// TwinCAT 3 PLC project _3d_printer
// ProgramVersion: 3.1.4023.0
// libraries:
//   Tc2_MC2, * (Beckhoff Automation GmbH)
//   Tc2_NCI, * (Beckhoff Automation GmbH)
//   Tc2_NcKinematicTransformation, * (Beckhoff Automation GmbH)
//   Tc2_PlcInterpolation, * (Beckhoff Automation GmbH)
//   Tc2_Standard, * (Beckhoff Automation GmbH)
//   Tc2_System, * (Beckhoff Automation GmbH)
//   Tc3_Module, * (Beckhoff Automation GmbH)
// project tree:
//   / PlcTask.TcTTO
//   POUs/ FB_PowerChannel.TcPOU, MAIN.TcPOU
// real-time tasks:
//   TASK PlcTask: cycle T#10ms, priority 20, ADS port 350
// motion (NC):
//   TASK NC-Task 1 SAF: cycle T#2ms, priority 4, ADS port 501
//   TASK NC-Task 1 SVB: cycle T#10ms, priority 8, ADS port 511
//   AXIS axis xy 1 (id 1)
//     Dynamic: AccelerationMaximum=2000, DecelerationMaximum=2000, Acceleration=1000, Deceleration=1000
//     Velo: SlowManual=50, FastManual=100, Maximum=500
//     OtherSettings: AllowMotionCmdToSlave=true
//     encoder EncType=1
//       EncPara: ScaleFactorNumerator=40, ScaleFactorDenominator=12800
//         Inc: RefSoftSyncMask=#x0000ffff
//     drive DrvType=5
//       Analog: VeloReferenz=400, TorqueSetpointScale=10, ScaleFactorActTorque=0.1
//       TimeComp: TaskDelayCycles=1
//     controller CtrType=1
//       CtrPara: PriorControlFactor=1
//         Observer: BandWidth=20
//   AXIS axis xy 2 (id 2)
//     Dynamic: AccelerationMaximum=2000, DecelerationMaximum=2000, Acceleration=1000, Deceleration=1000
//     Velo: SlowManual=50, FastManual=100, Maximum=500
//     OtherSettings: AllowMotionCmdToSlave=true
//     encoder EncType=1
//       EncPara: ScaleFactorNumerator=40, ScaleFactorDenominator=12800
//         Inc: RefSoftSyncMask=#x0000ffff
//     drive DrvType=5
//       Analog: VeloReferenz=400, TorqueSetpointScale=10, ScaleFactorActTorque=0.1
//       TimeComp: TaskDelayCycles=1
//     controller CtrType=1
//       CtrPara: PriorControlFactor=1
//         Observer: BandWidth=20
//   AXIS Extruder (id 4)
//     Dynamic: AccelerationMaximum=100, DecelerationMaximum=100, Acceleration=100, Deceleration=100, Jerk=500
//     Velo: Maximum=10
//     OtherSettings: AllowMotionCmdToSlave=true
//     encoder EncType=1
//       EncPara: ScaleFactorNumerator=22.857, ScaleFactorDenominator=12800
//         Inc: RefSoftSyncMask=#x0000ffff
//     drive DrvType=5
//       Analog: VeloReferenz=5, TorqueSetpointScale=10, ScaleFactorActTorque=0.1
//       TimeComp: TaskDelayCycles=1
//     controller CtrType=1
//       CtrPara: PriorControlFactor=1
//         Observer: BandWidth=20
//   AXIS X axis (id 5)
//     Dynamic: AccelerationMaximum=2000, DecelerationMaximum=2000, Acceleration=1000, Deceleration=1000
//     Velo: SlowManual=50, FastManual=100, Maximum=500
//     OtherSettings: AllowMotionCmdToSlave=true
//     encoder EncType=1
//       EncPara: ScaleFactorNumerator=1, ScaleFactorDenominator=0.1
//     drive DrvType=5
//       Analog: VeloReferenz=500, TorqueSetpointScale=10, ScaleFactorActTorque=0.1
//       TimeComp: TaskDelayCycles=1
//     controller CtrType=1
//       CtrPara: PriorControlFactor=1
//         Observer: BandWidth=20
//   AXIS Z axis (id 3)
//     Dynamic: AccelerationMaximum=100, DecelerationMaximum=100, Acceleration=50, Deceleration=50, Jerk=1000
//     Velo: SlowManual=1, FastManual=5, Maximum=10
//     OtherSettings: AllowMotionCmdToSlave=true
//     encoder EncType=4
//       EncPara: ScaleFactorNumerator=8, ScaleFactorDenominator=12800, MaxCount=#x0000ffff
//         Inc: RefSoftSyncMask=#x0000ffff
//     drive DrvType=24
//       Analog: VeloReferenz=80, TorqueSetpointScale=10, ScaleFactorActTorque=0.1
//       TimeComp: TaskDelayCycles=1
//     controller CtrType=1
//       CtrPara: PriorControlFactor=1
//         Observer: BandWidth=20
//   AXIS Y axis (id 6)
//     Dynamic: AccelerationMaximum=2000, DecelerationMaximum=2000, Acceleration=1000, Deceleration=1000
//     Velo: SlowManual=50, FastManual=100, Maximum=500
//     OtherSettings: AllowMotionCmdToSlave=true
//     encoder EncType=1
//     drive DrvType=5
//       Analog: VeloReferenz=500, TorqueSetpointScale=10, ScaleFactorActTorque=0.1
//       TimeComp: TaskDelayCycles=1
//     controller CtrType=1
//       CtrPara: PriorControlFactor=1
//         Observer: BandWidth=20

CONFIGURATION _3d_printer
    RESOURCE PLC ON TwinCAT3
        TASK PlcTask(INTERVAL := T#10ms, PRIORITY := 20);
        PROGRAM MAIN WITH PlcTask : MAIN;
    END_RESOURCE
END_CONFIGURATION

// ---- POUs/MAIN.TcPOU
PROGRAM MAIN
VAR
	
	fbPower: FB_PowerChannel;
	runGCode: ItpEnableDefaultGCode;
	fbBuildGroup: CfgBuildExt3DGroup;
	fbLoadGCode: ItpLoadProgEx;
	fbStartGCode: ItpStartStopEx;
	fbConfirmHsk: ItpConfirmHsk;
	//getSParam :ItpGetSParam;
	
	fbConfigKinGroup: FB_KinConfigGroup;
    stAxesConfig: ST_KinAxes;
	in_stKinToPlc AT %I*  : NCTOPLC_NCICHANNEL_REF;
	
	Xaxis: AXIS_REF;
	Yaxis: AXIS_REF;
	Zaxis: AXIS_REF;
	Extruder: AXIS_REF;
	XY_1: AXIS_REF;
	XY_2: AXIS_REF;

	Xhome: MC_Home;
	Yhome: MC_Home;
	Zhome: MC_Home;
	
	Xjog: MC_Jog;
	Yjog: MC_Jog;
	
	HomingSensorX AT %I*: BOOL;
	HomingSensorY AT %I*: BOOL;
	HomingSensorZ AT %I*: BOOL;
	
	
	in_stNciToPlc AT %I*: NCTOPLC_NCICHANNEL_REF;
	out_stPlcToNci AT %Q*: PLCTONC_NCICHANNEL_REF;
	
	
	State: INT;
	bConfirmHsk: BOOL := FALSE;
	sPrgName: STRING(255) := 'test.txt';
	nInterpreterState: UDINT;
	
	bEnable: BOOL := TRUE;
END_VAR


fbPower(
	bEnable:=bEnable, 
	fOvr:= 100.0, 
	stX:=Xaxis, 
	stY:=Yaxis, 
	stZ:=Zaxis,
	stXY_1:= XY_1,
	stXY_2:= XY_2,
	stPlcToNci:=out_stPlcToNci , 
	bAllAxesReady=> );
	

	
CASE State OF
	0: // init
	
	IF fbPower.bAllAxesReady THEN
		State := 10; 
	END_IF
	
	10:
	
	stAxesConfig.nAxisIdsAcs[1] := XY_2.NcToPlc.AxisId;
	stAxesConfig.nAxisIdsAcs[2] := XY_1.NcToPlc.AxisId;
	stAxesConfig.nAxisIdsMcs[1] := Xaxis.NcToPlc.AxisId;
	stAxesConfig.nAxisIdsMcs[2] := Yaxis.NcToPlc.AxisId;
	
	fbConfigKinGroup(
    bExecute       := TRUE ,
    bCartesianMode := TRUE ,
    stAxesList     := stAxesConfig,
    stKinRefIn     := in_stKinToPlc );
	
	IF NOT fbConfigKinGroup.bBusy THEN
		IF NOT fbConfigKinGroup.bError THEN
			State:=20;
		END_IF
	END_IF
	20:
	Xjog(Axis:= Xaxis,JogBackwards:= TRUE , Velocity:= 0.01, Deceleration:= 1500);
	IF NOT HomingSensorX THEN
		Xjog(Axis:= Xaxis,JogBackwards:= FALSE);
		//State:=21;
	END_IF
	
	21:
	Yjog(Axis:= Yaxis,JogBackwards:= TRUE , Velocity:= 0.01, Deceleration:= 1500);
	IF NOT HomingSensorY THEN
		Yjog(Axis:= Yaxis,JogBackwards:= FALSE);
		
		//State:=21;
	END_IF
	
	22:
	Zhome(axis := Zaxis,execute := TRUE,BCalibrationCam := NOT HomingSensorZ);
	IF Zhome.Done THEN
		//State:=30;
	END_IF
	
	30:
	
	fbLoadGCode(
		sNciToPlc:=in_stNciToPlc, 
		bExecute:=TRUE, 
		sPrg:= sPrgName, 
		nLength:= INT_TO_UDINT(LEN(sPrgName)), 
		tTimeOut:= , 
		bBusy=> , 
		bErr=> , 
		nErrId=> );
	IF NOT fbLoadGCode.bBusy THEN
		IF NOT fbLoadGCode.bErr THEN
			fbLoadGCode(sNciToPlc:=in_stNciToPlc, bExecute:=FALSE); 
			State	:= 40;				
		END_IF
	END_IF
	40:
	
	nInterpreterState	:= ItpGetStateInterpreter(sNciToPlc:=in_stNciToPlc);
	IF nInterpreterState = Tc2_NCI.NCI_INTERPRETER_READY THEN
		State	:= 50;		
	END_IF
	50:
	fbBuildGroup(
		bExecute:=TRUE,
		nGroupId:=ItpGetGroupId(sNciToPlc:=in_stNciToPlc),
		nXAxisId:=XAxis.NcToPlc.AxisId,
		nYAxisId:=YAxis.NcToPlc.AxisId,
		nZAxisId:=ZAxis.NcToPlc.AxisId,
		tTimeOut:=T#2S );
		
	IF NOT fbBuildGroup.bBusy THEN
		fbBuildGroup( bExecute:=FALSE );
		
		IF NOT fbBuildGroup.bErr THEN
			State	:= 30;
		END_IF
	END_IF

	
	60:
	
	// start g-code file
	fbStartGCode(
		bStart:=TRUE, 
		bStop:=FALSE, 
		tTimeOut:= , 
		sNciToPlc:= in_stNciToPlc, 
		bBusy=> , 
		bErr=> , 
		nErrId=> );
	IF NOT fbStartGCode.bBusy THEN
		IF NOT fbStartGCode.bErr THEN
			State	:= 60;			
		END_IF
		fbStartGCode( bStart:=FALSE, sNciToPlc:= in_stNciToPlc ); 
	END_IF
	70: //during print
	
	END_CASE

END_PROGRAM

// ---- POUs/FB_PowerChannel.TcPOU
FUNCTION_BLOCK FB_PowerChannel
VAR_INPUT
	bEnable			: BOOL := FALSE;
	fOvr			: LREAL;
END_VAR
VAR_IN_OUT
	stX				: AXIS_REF;
	stY 			: AXIS_REF;
	stZ				: AXIS_REF;
	stPlcToNci		: PLCTONC_NCICHANNEL_REF;
END_VAR
VAR_OUTPUT
	bAllAxesReady	: BOOL := FALSE;
END_VAR
VAR
	fbPowerX		:	MC_Power;
	fbPowerY		:	MC_Power;
	fbPowerZ		:	MC_Power;
END_VAR

fbPowerX(
	Axis:=stX , 
	Enable:=bEnable , 
	Enable_Positive:= bEnable, 
	Enable_Negative:= bEnable, 
	Override:=fOvr , 
	BufferMode:= , 
	Status=> , 
	Busy=> , 
	Active=> , 
	Error=> , 
	ErrorID=> );
fbPowerY(
	Axis:=stY , 
	Enable:=bEnable , 
	Enable_Positive:= bEnable, 
	Enable_Negative:= bEnable, 
	Override:=fOvr , 
	BufferMode:= , 
	Status=> , 
	Busy=> , 
	Active=> , 
	Error=> , 
	ErrorID=> );
fbPowerZ(
	Axis:=stZ , 
	Enable:=bEnable , 
	Enable_Positive:= bEnable, 
	Enable_Negative:= bEnable, 
	Override:=fOvr , 
	BufferMode:= , 
	Status=> , 
	Busy=> , 
	Active=> , 
	Error=> , 
	ErrorID=> );	
	
ItpSetOverridePercent(fOverridePercent:=fOvr, sPlcToNci:=stPlcToNci);

IF fbPowerX.Status AND fbPowerY.Status AND fbPowerZ.Status THEN
	bAllAxesReady	:= TRUE;
ELSE
	bAllAxesReady	:= FALSE;
END_IF

END_FUNCTION_BLOCK
